// TIA Portal V21 export
ORGANIZATION_BLOCK "OB_INSTRUMENTOS"   // OB130, LAD, ProgramCycle
TITLE = OB_INSTRUMENTOS
{ S7_Optimized_Access := 'TRUE' }
VERSION : 0.1
// stored: AutoNumber true, IsIECCheckEnabled false, SetENOAutomatically false
   VAR_INPUT
      Initial_Call : Bool;
      Remanence : Bool;
   END_VAR
BEGIN
END_ORGANIZATION_BLOCK
